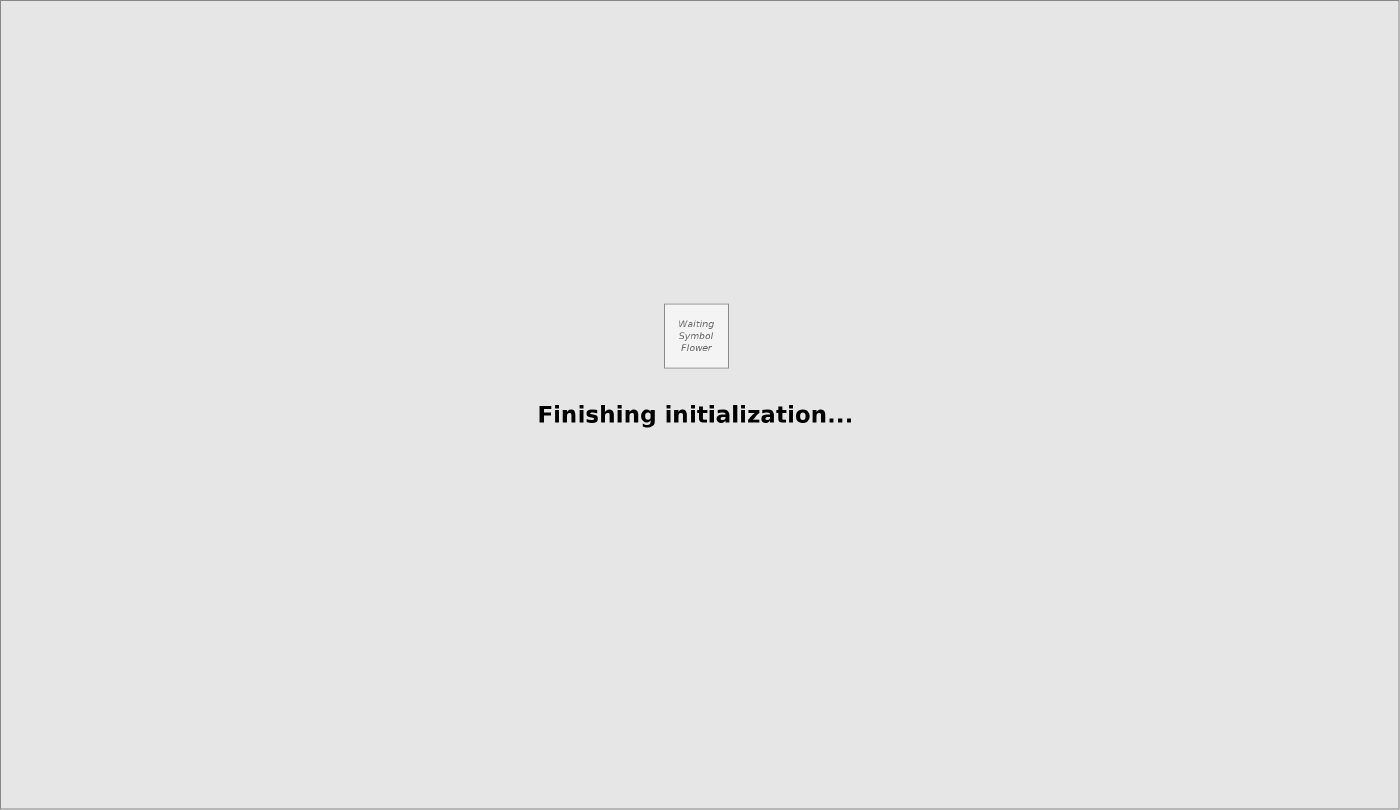
VISUALIZATION PageReadyInitialized  // 1520x880
    WaitingSymbolFlower (721,330 70x70)
    Label (530,430 450x40), "Finishing initialization..."
END_VISUALIZATION

(* stored: Version 1.1.0.1, ProductVersion 3.1.4024.9
   Visu PageReadyInitialized: Id {9102d4b5-7eac-440f-b5c8-dba014dcc8e6} *)
